TYPE unMyINT :
UNION
	nINT	: INT;
	nSINT	: ARRAY[1..2] OF SINT;
END_UNION
END_TYPE

(* stored: Version 1.1.0.1, ProductVersion 3.1.4024.12
   DUT unMyINT: Id {ca7b7b2f-9601-4c9b-be4e-5ca2502736c8} *)
